# EPICS substitutions: current/app/Db/inficon.substitutions
file inficon.template
{
    pattern
    { DEV,      PORT,       CSCAN,     DSCAN    }
    { $(DEV),   $(PORT),    $(CSCAN),  $(DSCAN) }
}
